(* PLC project fbd_arith, plcc plcc tests 1 *)
(* stored: creationDateTime 2026-09-27T00:00:00 *)

FUNCTION Scale : DINT
  VAR_INPUT
    x : DINT;
    k : DINT;
    ofs : DINT;
  END_VAR
  VAR  (* added by the conversion: wires and edge detectors of the diagram *)
    _MUL4_OUT : DINT;
    _ADD5_OUT : DINT;
  END_VAR

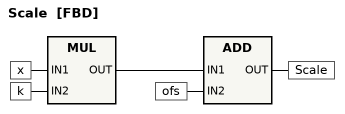
(* FBD diagram, written out as Structured Text *)
_MUL4_OUT := x * k;
_ADD5_OUT := _MUL4_OUT + ofs;
Scale := _ADD5_OUT;
END_FUNCTION

FUNCTION_BLOCK Integrator
  VAR_INPUT
    x : DINT;
  END_VAR
  VAR_OUTPUT
    total : DINT;
  END_VAR
  VAR  (* added by the conversion: wires and edge detectors of the diagram *)
    _ADD3_OUT : DINT;
  END_VAR

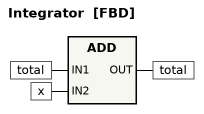
(* FBD diagram, written out as Structured Text *)
_ADD3_OUT := total + x;
total := _ADD3_OUT;
END_FUNCTION_BLOCK

PROGRAM Calc
  VAR
    a : DINT;
    b : DINT;
    c : DINT;
    y : DINT;
    s : DINT;
    m : DINT;
    lim : DINT;
    sc : DINT;
    agtb : BOOL;
    flag : BOOL;
    other : BOOL;
    both : BOOL;
    tot : DINT;
    integ : Integrator;
  END_VAR
  VAR  (* added by the conversion: wires and edge detectors of the diagram *)
    _ADD4_OUT : DINT;
    _MUL5_OUT : DINT;
    _MAX12_OUT : DINT;
    _LIMIT17_OUT : DINT;
    _Scale22_OUT : DINT;
    _GT26_OUT : BOOL;
    _AND30_OUT : BOOL;
  END_VAR

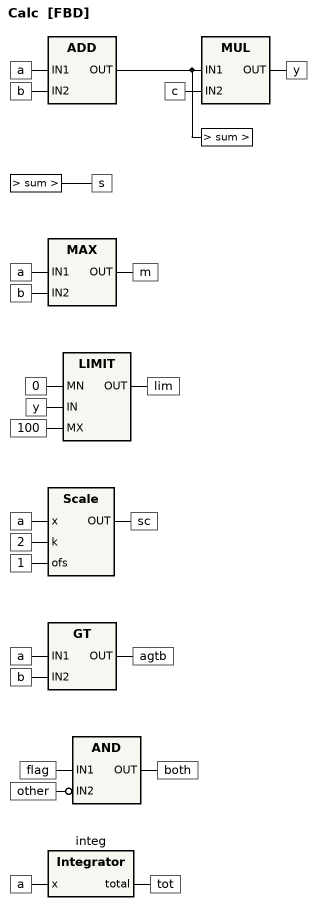
(* FBD diagram, written out as Structured Text *)
_ADD4_OUT := a + b;
_MUL5_OUT := _ADD4_OUT * c;
y := _MUL5_OUT;
s := _ADD4_OUT;
_MAX12_OUT := MAX(a, b);
m := _MAX12_OUT;
_LIMIT17_OUT := LIMIT(0, y, 100);
lim := _LIMIT17_OUT;
_Scale22_OUT := Scale(a, 2, 1);
sc := _Scale22_OUT;
_GT26_OUT := a > b;
agtb := _GT26_OUT;
_AND30_OUT := flag AND NOT other;
both := _AND30_OUT;
integ(x := a);
tot := integ.total;
END_PROGRAM
